// TwinCAT 3 PLC project Untitled3
// ProgramVersion: 3.1.4026.21
// libraries:
//   Tc2_Standard, * (Beckhoff Automation GmbH)
//   Tc2_System, * (Beckhoff Automation GmbH)
//   Tc3_EventLogger, * (Beckhoff Automation GmbH)
// project tree:
//   DUTs/ enBufferStatus.TcDUT, E_DeviceStatus.TcDUT, E_MotorStatus.TcDUT, enPalletStackerStatus.TcDUT
//   Interfaces/ ITFGesimuleerdDI.TcIO, ITFGesimuleerdDO.TcIO, ITFGesimuleerdAI.TcIO, ITFGesimuleerdAO.TcIO, ITFPalletStacker.TcIO, ITFServoMotor.TcIO, Temp_ITFLoopband.TcIO, Temp_ITFPalletPins.TcIO
//   / PlcTask.TcTTO
//   POUs/FB/ fbAfstandSensor.TcPOU, fbControllerPalletStacker.TcPOU, fbLichtSensor.TcPOU, fbPalletStacker.TcPOU, fbStackerServo.TcPOU, fbTemploopband.TcPOU, fbTemppalletpins.TcPOU
//   POUs/ MAIN.TcPOU
// real-time tasks:
//   TASK PlcTask: cycle T#10ms, priority 20, ADS port 350

CONFIGURATION Untitled3
    RESOURCE PLC ON TwinCAT3
        TASK PlcTask(INTERVAL := T#10ms, PRIORITY := 20);
        PROGRAM MAIN WITH PlcTask : MAIN;
    END_RESOURCE
END_CONFIGURATION

// ---- DUTs/enBufferStatus.TcDUT
{attribute 'qualified_only'}
{attribute 'strict'}
{attribute 'to_string'}
TYPE enBufferStatus :
(
	Leeg := 0,
	DeelsGevuld := 1,
	BijnaVol := 2,
	vol:= 3
);
END_TYPE

// ---- DUTs/E_DeviceStatus.TcDUT
{attribute 'qualified_only'}
{attribute 'strict'}
{attribute 'to_string'}
TYPE E_DeviceStatus :
(
	Uit := 0,
	Aan := 1,
	Error:= 2
);
END_TYPE

// ---- DUTs/E_MotorStatus.TcDUT
{attribute 'qualified_only'}
{attribute 'strict'}
{attribute 'to_string'}
TYPE E_MotorStatus :
(
	Uit := 0,
	Aan := 1,
	Error:= 2,
	Optoeren:= 3,
	Aftoeren:= 4
);
END_TYPE

// ---- DUTs/enPalletStackerStatus.TcDUT
{attribute 'qualified_only'}
{attribute 'strict'}
{attribute 'to_string'}
TYPE enPalletStackerStatus :
(
	Idle := 0,
	Collecting:= 1,
	PinsUitBewegen:= 2,
	LiftBewegen:= 3,
	Omwisselen:= 4,
	Legen:= 5,
	Error:= 6,
	PalletLaden:= 7,
	PinsInBewegen:= 8
);
END_TYPE

// ---- Interfaces/ITFGesimuleerdDI.TcIO
INTERFACE ITFGesimuleerdDI

PROPERTY SensorWaarde : bool
GET
END_GET
SET
END_SET
END_PROPERTY

END_INTERFACE

// ---- Interfaces/ITFGesimuleerdDO.TcIO
INTERFACE ITFGesimuleerdDO

PROPERTY SensorWaarde : bool
GET
END_GET
SET
END_SET
END_PROPERTY

END_INTERFACE

// ---- Interfaces/ITFGesimuleerdAI.TcIO
INTERFACE ITFGesimuleerdAI

PROPERTY SensorWaarde : int
GET
END_GET
SET
END_SET
END_PROPERTY

END_INTERFACE

// ---- Interfaces/ITFGesimuleerdAO.TcIO
INTERFACE ITFGesimuleerdAO

PROPERTY SensorWaarde : int
GET
END_GET
SET
END_SET
END_PROPERTY

END_INTERFACE

// ---- Interfaces/ITFPalletStacker.TcIO
INTERFACE ITFPalletStacker

METHOD CollectPallet : bool
VAR_INPUT
END_VAR
END_METHOD

METHOD EmptyStack : bool
VAR_INPUT
END_VAR
END_METHOD

METHOD Reset
VAR_INPUT
END_VAR
END_METHOD

METHOD StackPallet : bool
VAR_INPUT
END_VAR
END_METHOD

PROPERTY Status : E_DeviceStatus
GET
END_GET
SET
END_SET
END_PROPERTY

METHOD Stop
VAR_INPUT
END_VAR
END_METHOD

END_INTERFACE

// ---- Interfaces/ITFServoMotor.TcIO
INTERFACE ITFServoMotor

METHOD BeweegNaarDoel
VAR_INPUT
END_VAR
END_METHOD

PROPERTY DoelPositie : int
GET
END_GET
SET
END_SET
END_PROPERTY

PROPERTY Enable : bool
GET
END_GET
SET
END_SET
END_PROPERTY

PROPERTY MotorStatus : E_motorstatus
GET
END_GET
SET
END_SET
END_PROPERTY

PROPERTY Positie : int
GET
END_GET
END_PROPERTY

END_INTERFACE

// ---- Interfaces/Temp_ITFLoopband.TcIO
INTERFACE Temp_ITFLoopband

METHOD Beweeg
VAR_INPUT
END_VAR
END_METHOD

METHOD BeweegInLift
VAR_INPUT
END_VAR
END_METHOD

METHOD Stop
VAR_INPUT
END_VAR
END_METHOD

END_INTERFACE

// ---- Interfaces/Temp_ITFPalletPins.TcIO
INTERFACE Temp_ITFPalletPins

METHOD ErinBewegen :bool
VAR_INPUT
END_VAR
END_METHOD

METHOD EruitBewegen :BOOL
VAR_INPUT
END_VAR
END_METHOD

END_INTERFACE

// ---- POUs/MAIN.TcPOU
PROGRAM MAIN
VAR
StackerMotor : fbStackerServo();
PalletStacker : fbPalletStacker();
Ctrl : fbControllerPalletStacker;

bDeur1Dicht : BOOL := 1;
bDeur2Dicht : BOOL:= 1;
bNoodstop    : BOOL:= 0;

    iStackerOperatie : INT := 0;
	fbLoopband : fbTemploopband;
    fbPins     : fbTemppalletpins;
    fbLift     : fbStackerServo;
    fbAfstandSensor  : fbAfstandSensor;
	fbPalletBufferSensor : fbLichtSensor;
	fbPalletInLiftSensor : fbLichtSensor;
END_VAR

// Decode tester buttons into one‑shot commands
Ctrl.bCmdCollect := (iStackerOperatie = 1);
Ctrl.bCmdLegen   := (iStackerOperatie = 2);

// Call controller FB
Ctrl(
    fbStacker := palletstacker,
    bDeur1Dicht := bDeur1Dicht,
    bDeur2Dicht := bDeur2Dicht,
    bNoodstop := bNoodstop,
);

// reset tester after issuing the command
IF iStackerOperatie <> 0 THEN
   iStackerOperatie := 0;
END_IF

END_PROGRAM

// ---- POUs/FB/fbStackerServo.TcPOU
FUNCTION_BLOCK fbStackerServo implements ITFServoMotor
VAR_INPUT
END_VAR
VAR_OUTPUT
END_VAR
VAR
	
	IPositie : INT;
	TONBeweegTimer : TON;
	BTONVariabele : BOOL;
	EMotorStatusIntern : E_MotorStatus;
	IDoelPositie	: INT;
	BInternEnable : BOOL;
	
	MotorStatusString: STRING;
END_VAR

MotorStatusString := TO_STRING(EMotorStatusIntern);

METHOD PUBLIC BeweegNaarDoel
VAR_INPUT

END_VAR

VAR CONSTANT
	IMotorSnelheid : INT := 1; 
	IMotorStopSnelheid : INT:= 5;
END_VAR

//notes
//  status schrijven en
VAR
	BBewegenActief: BOOL;
END_VAR
(* ================= TIMER ================= *)
TONBeweegTimer(
    IN := BInternEnable AND NOT BBewegenActief,
    PT := T#0.3S
);

(* ================= START NA TIMER ================= *)
IF TONBeweegTimer.Q THEN
    BBewegenActief := TRUE;
    TONBeweegTimer(IN := FALSE);   // DIRECT reset → cruciaal
END_IF

(* ================= STATUS ================= *)
IF BInternEnable THEN
    EMotorStatusIntern := 1;
ELSE
    EMotorStatusIntern := 0;
END_IF

(* ================= BEWEGEN ================= *)
IF BInternEnable AND BBewegenActief THEN

    IF IDoelPositie > IPositie THEN
        IPositie := IPositie + IMotorSnelheid;
        EMotorStatusIntern := 3;

        IF IPositie >= IDoelPositie THEN
            IPositie := IDoelPositie;
            BBewegenActief := FALSE;
        END_IF

    ELSIF IDoelPositie < IPositie THEN
        IPositie := IPositie - IMotorSnelheid;
        EMotorStatusIntern := 4;

        IF IPositie <= IDoelPositie THEN
            IPositie := IDoelPositie;
            BBewegenActief := FALSE;
        END_IF

    ELSE
        BBewegenActief := FALSE;
    END_IF
END_IF

(* ================= UIT / STOP ================= *)
IF NOT BInternEnable THEN
    BBewegenActief := FALSE;
    TONBeweegTimer(IN := FALSE);

    IF IPositie > 0 THEN
        IPositie := IPositie - IMotorStopSnelheid;
        IF IPositie < 0 THEN IPositie := 0; END_IF

    ELSIF IPositie < 0 THEN
        IPositie := IPositie + IMotorStopSnelheid;
        IF IPositie > 0 THEN IPositie := 0; END_IF
    END_IF
END_IF
END_METHOD

PROPERTY DoelPositie : int
GET
doelpositie := idoelpositie;
END_GET
SET
idoelpositie := doelpositie;
END_SET
END_PROPERTY

PROPERTY Enable : bool
GET
Enable := BInternEnable;
END_GET
SET
BInternEnable:= Enable;
END_SET
END_PROPERTY

PROPERTY MotorStatus : E_MotorStatus
GET
MotorStatus:=  EMotorStatusIntern;
END_GET
SET
EMotorStatusIntern := MotorStatus;
END_SET
END_PROPERTY

PROPERTY Positie : INT
GET
positie:= IPositie;
END_GET
END_PROPERTY

END_FUNCTION_BLOCK

// ---- POUs/FB/fbPalletStacker.TcPOU
FUNCTION_BLOCK fbPalletStacker IMPLEMENTS ITFGesimuleerdAO, ITFPalletStacker
VAR_INPUT
bDeurDicht           : BOOL;  // Safety door switch (TRUE = closed/safe)
bNoodstopOk    : BOOL;
bVeiligheidHold : BOOL;
END_VAR
VAR_OUTPUT
	bPalletError :bool := 0;
END_VAR

VAR CONSTANT
	iMaxPallet : UINT := 5;
	ipallethoogte : UINT := 20;
	iplatformhoogte : UINT := 0;
	iMaxPalletSensor : UINT:= (iMaxPallet * ipallethoogte + iplatformhoogte);
END_VAR

VAR	
	bRunPermit  : BOOL; 
	EStatusVoorError : enPalletStackerStatus;
	bLegenDone        : BOOL;
	bDeurMagOpen      : BOOL;  // HMI indicator
	bLegenConfirmed       : BOOL;  // HMI confirmation after emptying
	
	StartCmd             : BOOL;  // HMI start cycle
	StopCmd              : BOOL;  // HMI stop cycle
	CycleActive          : BOOL;  // internal running flag
	
	ClearForLoad         : BOOL;  // internal gating
	liftTol              : REAL;  // position tolerance

	fbLoopband : fbTemploopband;
    fbPins     : fbTemppalletpins;
    fbLift     : fbStackerServo;
    fbAfstandSensor  : fbAfstandSensor;
	fbPalletBufferSensor : fbLichtSensor;
	fbPalletInLiftSensor : fbLichtSensor;

    fbStackerStatus    : enPalletStackerStatus := enPalletStackerStatus.Idle;
	fbStatusString : string;

	ePalletBufferStatus : enBufferStatus := 0;
	
	sVolgendeStap :STRING;
	bError: BOOL;
	bKlaarVoorVolgende: BOOL := 1;
	
	tonErrorTimer: TON;
	
	tiHmiTimer: TIME;
	bAlarmAck: BOOL;
	bAlarmTrig: BOOL;
	bPalletVoorLiftSensor: BOOL;
	sbuffervol: STRING;
	bStatusVeranderd: BOOL;
	eVorigeStatus: enPalletStackerStatus;
	
	fblogger : FB_TcEventLogger;
	fbalarm : FB_tcalarm;
	fbsource: FB_tcsourceinfo;
	fbargument: fb_tcarguments;

	bDeurSlot: BOOL;
END_VAR

// Update bufferstatus
fbStatusString := TO_STRING(fbStackerStatus);
sbuffervol := TO_STRING(ePalletBufferStatus);
tiHmiTimer := tonErrorTimer.ET;

// Run permit from controller safety
bRunPermit := bNoodstopOk AND (NOT bVeiligheidHold);

// Detect state change for timer reset
bStatusVeranderd := (fbStackerStatus <> eVorigeStatus);
IF bStatusVeranderd THEN
    eVorigeStatus := fbStackerStatus;
    bAlarmTrig := FALSE;
END_IF

// Safety interlock (EStop or SafetyHold)
IF NOT bRunPermit THEN
    fbLoopband.Stop();
    fbLift.Enable := 0;
    bAlarmTrig := FALSE;
	
	fbsource.Clear();
	fbsource.sName := 'Noodstop';
	fbalarm.CreateEx(tc_events.StackerEvents.Noodstop, TRUE, fbsource);
	fbalarm.Raise(0);
ELSE
    fbLift.Enable := 1;
END_IF

// ErrorTimer handling (reset on state change or safety)
IF bStatusVeranderd OR NOT bAlarmTrig OR NOT bRunPermit OR NOT bDeurDicht THEN
    tonErrorTimer(IN := FALSE, PT := T#60S);
ELSE
    tonErrorTimer(IN := TRUE, PT := T#60S);
END_IF

IF tonErrorTimer.Q AND fbStackerStatus <> enPalletStackerStatus.Error THEN
    EStatusVoorError := fbStackerStatus;
    fbStackerStatus := enPalletStackerStatus.Error;
    bAlarmTrig := FALSE;
	
	fbsource.Clear();
	fbsource.sName := 'error timer';
	fbalarm.CreateEx(tc_events.StackerEvents.Vastgelopen, TRUE, fbsource);
	// hoe kijk je als dit gebeurt
	fbalarm.Raise(0);
	
END_IF

// Bufferstatus bepalen
IF fbAfstandSensor.SensorWaarde >= iMaxPalletSensor THEN
    ePalletBufferStatus := enBufferStatus.vol;
ELSIF fbAfstandSensor.SensorWaarde = iMaxPalletSensor - 2 * ipallethoogte
      AND iMaxPalletSensor > 2 * ipallethoogte + iplatformhoogte THEN
    ePalletBufferStatus := enBufferStatus.BijnaVol;
ELSIF fbAfstandSensor.SensorWaarde >= iplatformhoogte + ipallethoogte THEN
    ePalletBufferStatus := enBufferStatus.DeelsGevuld;
ELSE
    ePalletBufferStatus := enBufferStatus.Leeg;
END_IF

// Clear to load condition: no pins out, lift at load height, not mid-cycle
ClearForLoad :=
    (NOT fbPins.PinsUit)
    AND (ABS(fbLift.positie - (iplatformhoogte + ipallethoogte)) <= liftTol)
    AND (NOT bPalletVoorLiftSensor);

// Door lock logic
IF NOT bRunPermit THEN
    bDeurSlot := FALSE;
ELSIF fbStackerStatus = enPalletStackerStatus.Legen THEN
    IF bLegenDone THEN
        bDeurSlot := FALSE;
    ELSE
        bDeurSlot := TRUE;
    END_IF
ELSIF CycleActive THEN
    bDeurSlot := TRUE;
ELSE
    bDeurSlot := FALSE;
END_IF

bDeurMagOpen := NOT bDeurSlot;

// Start/Stop behavior
IF StopCmd THEN
    CycleActive := FALSE;
END_IF

//IF StartCmd AND bDeurDicht AND bRunPermit THEN
   // CycleActive := TRUE;
//END_IF

CASE fbStackerStatus OF
//==================== Idle ====================
enPalletStackerStatus.Idle:
    sVolgendeStap := 'Idle: wacht op start/legen';
    bKlaarVoorVolgende := FALSE;
    bPalletVoorLiftSensor := 0;
    bAlarmTrig := FALSE;
    bLegenDone := FALSE;

    //IF CycleActive THEN
      //  State := E_PalletStackerStatus.Collecting;
    //END_IF

//==================== Collecting ====================
enPalletStackerStatus.Collecting:
    sVolgendeStap := 'Collecting: pallet naar buffer';

    IF NOT bRunPermit THEN
        sVolgendeStap := 'Collecting: veiligheidsstop, pauze';
        fbLoopband.Stop();
        bAlarmTrig := FALSE;

    ELSIF NOT bDeurDicht THEN
        sVolgendeStap := 'Collecting: deur open, pauze';
        fbLoopband.Stop();
        bAlarmTrig := FALSE;
		
		fbsource.Clear();
		fbsource.sName := 'deur open';
		fbalarm.CreateEx(tc_events.StackerEvents.Door1Open, TRUE, fbsource);
	    fbalarm.Raise(0);
		
    // 1) Breng pallet naar voor de lift
    ELSIF (ePalletBufferStatus = enBufferStatus.Leeg OR ePalletBufferStatus = enBufferStatus.DeelsGevuld)
          AND NOT bPalletVoorLiftSensor THEN

        fbLoopband.Beweeg();
        sVolgendeStap := 'Collecting: wacht op PalletBeforeLiftSensor';

        IF fbPalletBufferSensor.SensorWaarde1 THEN
            fbLoopband.Stop();
            bPalletVoorLiftSensor := 1;
            bAlarmTrig := FALSE;
        ELSE
            bAlarmTrig := TRUE;
        END_IF
		


    // 2) Zorg dat lift klaar is (geen pins uit, juiste hoogte)
    ELSIF bPalletVoorLiftSensor AND NOT bKlaarVoorVolgende THEN
        IF NOT fbPins.pinsin THEN
            fbPins.ErinBewegen();
            sVolgendeStap := 'Collecting: pins in voor laden';
            bAlarmTrig := TRUE;
        ELSE
            fbLift.DoelPositie := iplatformhoogte + ipallethoogte;
            fbLift.BeweegNaarDoel();
            sVolgendeStap := 'Collecting: lift naar laadhoogte';

            IF ABS(fbLift.positie - (iplatformhoogte + ipallethoogte)) <= liftTol THEN
                bKlaarVoorVolgende := TRUE;
                bAlarmTrig := FALSE;
            ELSE
                bAlarmTrig := TRUE;
            END_IF
        END_IF

    // 3) Pallet in lift laden
    ELSIF bKlaarVoorVolgende AND bPalletVoorLiftSensor THEN
        fbLoopband.Beweeg();
        sVolgendeStap := 'Collecting: wacht op PalletInLiftSensor';

        IF fbPalletInLiftSensor.SensorWaarde1 THEN
            bKlaarVoorVolgende := FALSE;
            bPalletVoorLiftSensor := 0;
            fbLoopband.Stop();
            fbStackerStatus := enPalletStackerStatus.PinsUitBewegen;
            bAlarmTrig := FALSE;
        ELSE
            bAlarmTrig := TRUE;
        END_IF
		

	
	ELSIF ePalletBufferStatus = enBufferStatus.vol OR ePalletBufferStatus = enBufferStatus.BijnaVol THEN
    fbLoopband.Stop();
    sVolgendeStap := 'Collecting: buffer vol, cyclus stopt';
    bAlarmTrig := FALSE;
    CycleActive := FALSE;
    fbStackerStatus := enPalletStackerStatus.Idle;
    END_IF

//==================== Pins Uit Bewegen ====================
enPalletStackerStatus.PinsUitBewegen:
    sVolgendeStap := 'PinsUit: pallet neerzetten op pins';

    IF NOT bRunPermit THEN
        sVolgendeStap := 'PinsUit: veiligheidsstop, pauze';
        bAlarmTrig := FALSE;
    ELSIF NOT bDeurDicht THEN
        sVolgendeStap := 'PinsUit: deur open, pauze';
        bAlarmTrig := FALSE;
    ELSIF fbPins.PinsUit THEN
        fbStackerStatus := enPalletStackerStatus.LiftBewegen;
        bAlarmTrig := FALSE;
    ELSE
        fbPins.EruitBewegen();
        bAlarmTrig := TRUE;
    END_IF

//==================== Lift Bewegen ====================
enPalletStackerStatus.LiftBewegen:
    sVolgendeStap := 'LiftBewegen: lift omlaag';

    IF NOT bRunPermit THEN
        sVolgendeStap := 'LiftBewegen: veiligheidsstop, pauze';
        bAlarmTrig := FALSE;
    ELSIF NOT bDeurDicht THEN
        sVolgendeStap := 'LiftBewegen: deur open, pauze';
        bAlarmTrig := FALSE;
    ELSIF fbPins.pinsuit THEN
        fbLift.DoelPositie := iplatformhoogte;
        fbLift.BeweegNaarDoel();

        IF ABS(fbLift.positie - iplatformhoogte) <= liftTol THEN
            fbStackerStatus := enPalletStackerStatus.PinsInBewegen;
            bAlarmTrig := FALSE;
        ELSE
            bAlarmTrig := TRUE;
        END_IF
    ELSE
        bAlarmTrig := TRUE;
    END_IF

//==================== Pins In Bewegen ====================
enPalletStackerStatus.PinsInBewegen:
    sVolgendeStap := 'PinsIn: pallet vrijgeven';

    IF NOT bRunPermit THEN
        sVolgendeStap := 'PinsIn: veiligheidsstop, pauze';
        bAlarmTrig := FALSE;
    ELSIF NOT bDeurDicht THEN
        sVolgendeStap := 'PinsIn: deur open, pauze';
        bAlarmTrig := FALSE;
    ELSIF fbPins.pinsin THEN
        fbStackerStatus := enPalletStackerStatus.PalletLaden;
        bAlarmTrig := FALSE;
    ELSE
        fbPins.ErinBewegen();
        bAlarmTrig := TRUE;
    END_IF

//==================== Pallet Laden ====================
enPalletStackerStatus.PalletLaden:
    sVolgendeStap := 'PalletLaden: lift omhoog klaar voor next';

    IF NOT bRunPermit THEN
        sVolgendeStap := 'PalletLaden: veiligheidsstop, pauze';
        bAlarmTrig := FALSE;
    ELSIF NOT bDeurDicht THEN
        sVolgendeStap := 'PalletLaden: deur open, pauze';
        bAlarmTrig := FALSE;
    ELSE
        fbLift.DoelPositie := iplatformhoogte + ipallethoogte;
        fbLift.BeweegNaarDoel();

        IF ABS(fbLift.positie - (iplatformhoogte + ipallethoogte)) <= liftTol THEN
            bKlaarVoorVolgende := TRUE;
            CycleActive := FALSE;
            fbStackerStatus := enPalletStackerStatus.Idle;
            fbAfstandSensor.SensorWaarde := fbAfstandSensor.SensorWaarde + ipallethoogte;
            bAlarmTrig := FALSE;
        ELSE
            bAlarmTrig := TRUE;
        END_IF
    END_IF

//==================== Legen ====================
enPalletStackerStatus.Legen:
    sVolgendeStap := 'Legen: pallets naar bodem';

    IF NOT bRunPermit THEN
        sVolgendeStap := 'Legen: veiligheidsstop, pauze';
        fbLoopband.Stop();
        bAlarmTrig := FALSE;

    ELSIF (NOT bDeurDicht) AND (NOT bLegenDone) THEN
        sVolgendeStap := 'Legen: deur open, pauze beweging';
        fbLoopband.Stop();
        bAlarmTrig := FALSE;
    ELSE
        IF NOT bLegenDone THEN
            fbLift.DoelPositie := 0;
            fbLift.BeweegNaarDoel();
            sVolgendeStap := 'Legen: lift naar bodem, pins uit';

            IF ABS(fbLift.positie - 0) <= liftTol THEN
                fbPins.EruitBewegen();
                IF fbPins.PinsUit THEN
                    bLegenDone := TRUE;
                    bAlarmTrig := FALSE;
                ELSE
                    bAlarmTrig := TRUE;
                END_IF
            ELSE
                bAlarmTrig := TRUE;
            END_IF
        ELSE
            sVolgendeStap := 'Legen: leeg, wacht confirm (deur mag open)';
            bAlarmTrig := FALSE;

            // Pas leeg teller na confirm en alleen als deur dicht
            IF bLegenConfirmed AND bDeurDicht THEN
                fbAfstandSensor.SensorWaarde := 0;
                bLegenDone := FALSE;
                fbStackerStatus := enPalletStackerStatus.Idle;
            END_IF
        END_IF
    END_IF

//==================== Error ====================
enPalletStackerStatus.Error:
    sVolgendeStap := 'ERROR: stop alles, wacht reset';
    bError := 1;
	

    fbLoopband.Stop();
    fbLift.Enable := 0;
    fbLift.DoelPositie := fbLift.positie;

    bKlaarVoorVolgende := FALSE;
    bPalletVoorLiftSensor := 0;
    bAlarmTrig := FALSE;
    CycleActive := FALSE;

    IF bAlarmAck = 1 THEN
        bError := 0;
        bAlarmTrig := FALSE;
        IF bDeurDicht THEN
            fbStackerStatus := EStatusVoorError;
        ELSE
            fbStackerStatus := enPalletStackerStatus.Idle;
        END_IF
    END_IF
END_CASE


IF (fbStackerStatus <> enPalletStackerStatus.Error) AND bDeurDicht AND bNoodstopOk AND NOT bVeiligheidHold THEN
    fbsource.Clear();
    fblogger.ClearAllAlarms();
END_IF

{warning 'Add method implementation '}
METHOD CollectPallet : bool
    IF fbStackerStatus = enPalletStackerStatus.idle AND NOT fbAfstandSensor.SensorWaarde >= iMaxPalletSensor THEN
        fbStackerStatus := enPalletStackerStatus.Collecting;
        CollectPallet := TRUE;
    ELSE
        CollectPallet := FALSE;
    END_IF
END_METHOD

{warning 'Add method implementation '}
METHOD EmptyStack : bool
    IF fbStackerStatus = enPalletStackerStatus.Idle AND NOT fbAfstandSensor.SensorWaarde >= iMaxPallet THEN
        fbStackerStatus := enPalletStackerStatus.Legen;
        EmptyStack := TRUE;
    ELSE
        EmptyStack := FALSE;
    END_IF
END_METHOD

{warning 'Add method implementation '}
METHOD Reset
END_METHOD

{warning 'Add property implementation'}
PROPERTY SensorWaarde : INT
GET
END_GET
SET
END_SET
END_PROPERTY

{warning 'Add method implementation '}
METHOD StackPallet : bool
    IF fbStackerStatus = enPalletStackerStatus.Idle AND NOT fbAfstandSensor.SensorWaarde >= iMaxPallet THEN
       // State := E_PalletStackerStatus.PinsBewegen;
        StackPallet := TRUE;
    ELSE
        StackPallet := FALSE;
    END_IF
END_METHOD

{warning 'Add property implementation'}
PROPERTY Status : E_DeviceStatus
GET
END_GET
SET
END_SET
END_PROPERTY

{warning 'Add method implementation '}
METHOD Stop
END_METHOD

END_FUNCTION_BLOCK

// ---- POUs/FB/fbTemploopband.TcPOU
FUNCTION_BLOCK fbTemploopband IMPLEMENTS temp_ITFloopband
VAR_INPUT
END_VAR
VAR_OUTPUT
END_VAR
VAR
	LoopbandActief : BOOL;
	
END_VAR

{warning 'Add method implementation '}
METHOD Beweeg
LoopbandActief:= 1;
END_METHOD

{warning 'Add method implementation '}
METHOD BeweegInLift
END_METHOD

{warning 'Add method implementation '}
METHOD Stop
LoopbandActief:= 0;
END_METHOD

END_FUNCTION_BLOCK

// ---- POUs/FB/fbTemppalletpins.TcPOU
FUNCTION_BLOCK fbTemppalletpins  IMPLEMENTS temp_ITFPalletPins
VAR_INPUT
END_VAR
VAR_OUTPUT
END_VAR
VAR
	PinsIn :BOOL:= FALSE;
	PinsUit :BOOL := TRUE;
	
END_VAR

{warning 'Add method implementation '}
METHOD Beweegpinsnaarbeneden : bool
END_METHOD

{warning 'Add method implementation '}
METHOD ErinBewegen : bool
END_METHOD

{warning 'Add method implementation '}
METHOD EruitBewegen : bool
END_METHOD

END_FUNCTION_BLOCK

// ---- POUs/FB/fbAfstandSensor.TcPOU
FUNCTION_BLOCK fbAfstandSensor IMPLEMENTS ITFGesimuleerdAO
VAR_INPUT
END_VAR
VAR_OUTPUT
END_VAR
VAR
	IHmiStackerAfstandSensorSim : INT;
END_VAR

{warning 'Add property implementation'}
PROPERTY SensorWaarde : INT
GET

SensorWaarde := IHmiStackerAfstandSensorSim;
END_GET
SET
IHmiStackerAfstandSensorSim:= SensorWaarde;
END_SET
END_PROPERTY

END_FUNCTION_BLOCK

// ---- POUs/FB/fbLichtSensor.TcPOU
FUNCTION_BLOCK fbLichtSensor IMPLEMENTS ITFGesimuleerdDO
VAR_INPUT
END_VAR
VAR_OUTPUT
END_VAR
VAR
	BHmiPalletSensorSim : BOOL;
	sensorwaarde1 : BOOL;
END_VAR

{warning 'Add property implementation'}
PROPERTY SensorWaarde : BOOL
GET
BHmiPalletSensorSim:= SensorWaarde1;
END_GET
SET
SensorWaarde1 := BHmiPalletSensorSim;
END_SET
END_PROPERTY

END_FUNCTION_BLOCK

// ---- POUs/FB/fbControllerPalletStacker.TcPOU
FUNCTION_BLOCK fbControllerPalletStacker
VAR_INPUT
    bCmdCollect     : BOOL;
    bCmdLegen       : BOOL;

    bDeur1Dicht    : BOOL;
    bDeur2Dicht    : BOOL;
    bNoodstop        : BOOL;

END_VAR

VAR_IN_OUT
    fbStacker           : fbPalletStacker(DoorClosed:= bDeur1Dicht); // change to your actual FB type
END_VAR

VAR_OUTPUT
    bVeiligheidsPauze  : BOOL;
    iActiveCmd     : INT;  
END_VAR
	
	VAR
	bAlleDeurenDicht : BOOL;
	bVeiligheidTrip      : BOOL;
	bVeiligheidsLatch     : BOOL;
	BVeiligheidAck       : BOOL; // HMI button
    rCollect : R_TRIG;
    rLegen   : R_TRIG;
    iCmdLatch : INT;

END_VAR

// Safety
bAlleDeurenDicht := bDeur1Dicht AND bDeur2Dicht;
bVeiligheidTrip := (NOT bAlleDeurenDicht) OR (bNoodstop);

IF bVeiligheidTrip THEN
    bVeiligheidsLatch := TRUE;
END_IF

IF BVeiligheidAck AND NOT bVeiligheidTrip THEN
    bVeiligheidsLatch := FALSE;
END_IF

bVeiligheidsPauze := bVeiligheidTrip OR bVeiligheidsLatch;

// Pass combined safety into stacker
fbStacker(
    bDeurDicht := bAlleDeurenDicht,
    bNoodstopOk := NOT bNoodstop,
    bVeiligheidHold := bVeiligheidsLatch
);

IF bVeiligheidsPauze THEN
    fbStacker.Stop();
    iCmdLatch := 0;
    iActiveCmd := 0;
END_IF

// Edge detect commands
rCollect(CLK := bCmdCollect);
rLegen(CLK := bCmdLegen);

IF rCollect.Q THEN iCmdLatch := 1; END_IF
IF rLegen.Q THEN
    //Stacker.EmptyStack();
    //ActiveCmd := 2;
    iCmdLatch := 0;
END_IF

// Execute commands
IF NOT bVeiligheidsPauze THEN
    // Empty has priority and can interrupt Collect
    IF rLegen.Q THEN
        fbStacker.EmptyStack();
        iActiveCmd := 2;
        iCmdLatch := 0;
    ELSIF iActiveCmd = 0 THEN
        IF iCmdLatch <> 0 THEN
            CASE iCmdLatch OF
                1: fbStacker.CollectPallet();
                2: fbStacker.EmptyStack();
            END_CASE
            iActiveCmd := iCmdLatch;
            iCmdLatch := 0;
        END_IF
    ELSE
        IF fbStacker.fbStackerStatus = enPalletStackerStatus.Idle THEN
            iActiveCmd := 0;
        END_IF
    END_IF
END_IF

END_FUNCTION_BLOCK
